PROGRAM MAIN
VAR
	M1: DUT_MotionStage;
	fbMotionStage: FB_MotionStage;
	nCounter: UINT;
END_VAR

fbMotionStage(stMotionStage:=M1);
nCounter := nCounter + 1;

END_PROGRAM

(* stored: Version 1.1.0.1, ProductVersion 3.1.4022.12
   POU MAIN: Id {9bcc2915-7068-448d-a348-931c17fac05a}, SpecialFunc None *)
